(* CoDeSys 2.3.9.62 project: Cap11_14.pro *)
(* Libraries: Standard.lib 2.6.14 10:37:46, IecSfc.lib 2.6.14 10:37:46 *)

(* Global variable list: Global_Variables *)
VAR_GLOBAL
       (* Entradas*)
	A:BOOL;
	B:BOOL;
      M:BOOL;
    	P:BOOL;
	E:BOOL;
	Rear:BOOL;
      (* Salidas*)
	MOTOR_IZ:BOOL;
	MOTOR_DE:BOOL;
	Funciona:BOOL;
       (* Para el simulador *)
	Vel:INT:=1;
END_VAR

(* POU PLC_PRG, ST *)
   PROGRAM PLC_PRG
VAR
END_VAR
Vehiculo();
END_PROGRAM

(* POU Vehiculo, ST *)
PROGRAM Vehiculo
VAR
	PosX: INT;
END_VAR
A:=FALSE;
B:=FALSE;


IF MOTOR_DE=TRUE THEN

     PosX:=PosX+Vel;

END_IF

IF MOTOR_IZ=TRUE THEN

     PosX:=PosX-Vel;

END_IF


IF PosX<=0 THEN
   A:=TRUE;
END_IF

IF PosX>=400 THEN
  B:=TRUE;
END_IF
END_PROGRAM

(* POU Automatismo, SFC *)
PROGRAM Automatismo
VAR
END_VAR
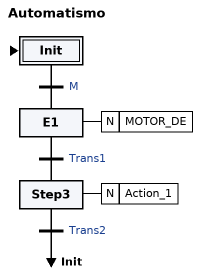
INITIAL_STEP Init:
END_STEP
TRANSITION FROM Init TO E1 := M;
END_TRANSITION
STEP E1:
	MOTOR_DE(N);
END_STEP
TRANSITION FROM E1 TO Step3 := Trans1;
END_TRANSITION
STEP Step3:
	Action_1(N);
END_STEP
TRANSITION FROM Step3 TO Init := Trans2;
END_TRANSITION
END_PROGRAM

(* POU MarchaParada, SFC *)
PROGRAM MarchaParada
VAR
END_VAR
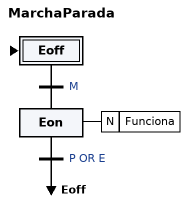
INITIAL_STEP Eoff:
END_STEP
TRANSITION FROM Eoff TO Eon := M;
END_TRANSITION
STEP Eon:
	Funciona(N);
END_STEP
TRANSITION FROM Eon TO Eoff := P OR E;
END_TRANSITION
END_PROGRAM

(* Visualisation Vehiculo
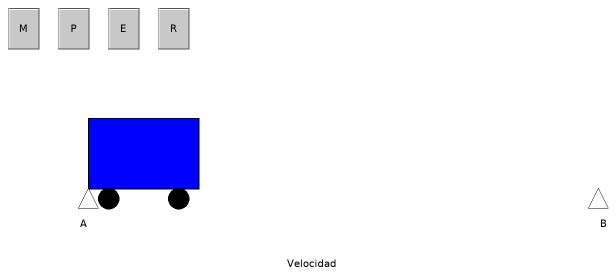
rectangle at (140,120)-(251,191): x offset Vehiculo.PosX
polygon at (130,190)-(150,210): alarm colour if .A
polygon at (640,190)-(660,210): alarm colour if .B
button at (60,10)-(91,51): text "M"; taps M
ellipse at (150,190)-(171,211): x offset Vehiculo.PosX
ellipse at (220,190)-(241,211): x offset Vehiculo.PosX
rectangle at (310,250)-(421,281): text "Velocidad"
rectangle at (80,210)-(191,241): text "A"
rectangle at (600,210)-(711,241): text "B"
button at (110,10)-(141,51): text "P"; taps P
button at (160,10)-(191,51): text "E"; taps E
button at (210,10)-(241,51): text "R"; taps Rear
1 elements of other kinds (tables, trends, ...) not read
*)
